{attribute 'linkalways'} 
{attribute 'no_explicit_call' := 'This FB is a CLASS and must be accessed using methods or properties'}
{attribute 'enable_dynamic_creation'}
FUNCTION_BLOCK Node_F_VN_AddContainers EXTENDS VisionNode
VAR
    ipSrcContainer1 : _ITcVnContainer;
    ipSrcContainer2 : _ITcVnContainer;
    ipDestContainer : _ITcVnContainer;
    hrPrev : _HRESULT(S_OK);
    hresult : _HRESULT(S_OK);
END_VAR

METHOD PUBLIC  Clone : I_Node
VAR
    pNode : POINTER TO Node_F_VN_AddContainers;
END_VAR
pNode := __NEW(Node_F_VN_AddContainers);
Clone := pNode^;
END_METHOD

METHOD FB_init : BOOL
VAR_INPUT
    bInitRetains : BOOL; // if TRUE, the retain variables are initialized (warm start / cold start)
    bInCopyCode : BOOL;  // if TRUE, the instance afterwards gets moved into the copy code (online change)
END_VAR
AddInput('ipSrcContainer1', ipSrcContainer1);
AddInput('ipSrcContainer2', ipSrcContainer2);
AddInput('hrPrev', hrPrev);
AddOutput('ipDestContainer', ipDestContainer);
AddOutput('hresult',hresult);
END_METHOD

METHOD PROTECTED OnExecute
hresult.Value := F_VN_AddContainers(
    ipSrcContainer1 := ipSrcContainer1.Value,
    ipSrcContainer2 := ipSrcContainer2.Value,
    ipDestContainer := ipDestContainer.Value,
    hrPrev:= hrPrev.Value);
END_METHOD

METHOD PUBLIC PreExecutionCheck
VAR_INPUT
    Check : I_PreExecutionChecks;
END_VAR
Check.IsTrue(ipSrcContainer1.IsValid, 'ipSrcContainer1 must be a valid container');
Check.IsTrue(ipSrcContainer2.IsValid, 'ipSrcContainer2 must be a valid container');
Check.IsTrue(ContainersHaveMatchingTypes(ipSrcContainer1.Value, ipSrcContainer2.Value), 'Source containers must have matching types');
Check.IsTrue(ContainersHaveMatchingNumberOfElements(ipSrcContainer1.Value, ipSrcContainer2.Value), 'Source containers must contain the same number of elements');
END_METHOD

END_FUNCTION_BLOCK

(* stored: Version 1.1.0.1, ProductVersion 3.1.4024.15
   POU Node_F_VN_AddContainers: Id {89ab1ec5-cf7a-0a84-0410-8f6cbee9e09c}, SpecialFunc None
   Folder Constructor: Id {fa866fd0-5198-0198-199a-f6f862f2e532}
   Method Clone: Id {9f7bcc86-7ee4-0b5d-0ca3-62069d0ac85f}
   Method FB_init: Id {4cd5091b-9fe0-00f1-18fc-f00dde0846a8}
   Method OnExecute: Id {b7f46372-b201-039a-0caa-acadecb782a1}
   Method PreExecutionCheck: Id {5deae83b-a123-0e04-01bd-c653fbe52d91} *)
